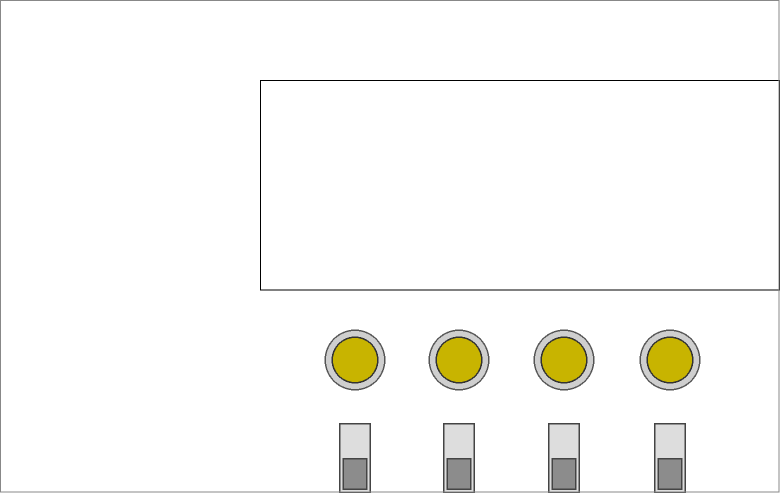
VISUALIZATION Visualization  // 780x493
    Rectangle (260,80 520x210)
    DipSwitch (320,423 70x70), variable: GVL.aSwitches[5], behaviour: TOGGLE, style: Switch-DipSwitch-Gray
    Lamp1 (320,325 70x70), variable: GVL.aLights[5], style: Lamp-Lamp1-Yellow
    DipSwitch (424,423 70x70), variable: GVL.aSwitches[6], behaviour: TOGGLE, style: Switch-DipSwitch-Gray
    Lamp1 (424,325 70x70), variable: GVL.aLights[6], style: Lamp-Lamp1-Yellow
    DipSwitch (529,423 70x70), variable: GVL.aSwitches[7], behaviour: TOGGLE, style: Switch-DipSwitch-Gray
    Lamp1 (529,325 70x70), variable: GVL.aLights[7], style: Lamp-Lamp1-Yellow
    DipSwitch (635,423 70x70), variable: GVL.aSwitches[8], behaviour: TOGGLE, style: Switch-DipSwitch-Gray
    Lamp1 (635,325 70x70), variable: GVL.aLights[8], style: Lamp-Lamp1-Yellow
END_VISUALIZATION

(* stored: Version 1.1.0.1, ProductVersion 3.1.4024.12
   Visu Visualization: Id {569d9c52-6f4a-4801-9b9c-c55cb942552c} *)
